FUNCTION_BLOCK FB_Roller_Door
VAR_INPUT
	// Inputs
    OpenBtn   : BOOL;
    CloseBtn  : BOOL;
    StopBtn   : BOOL;
    LS_Open   : BOOL;
    LS_Close  : BOOL;
END_VAR
VAR_OUTPUT
	// Outputs
    Motor_Up   : BOOL;
    Motor_Down : BOOL;
	Motor_Up_Reached:BOOL;
	Motor_Down_Reached:BOOL;
END_VAR
VAR
	// Internal states (latch)
    Opening : BOOL := FALSE;
    Closing : BOOL := FALSE;
END_VAR

// OPEN command
IF OpenBtn AND NOT LS_Open THEN
    Opening := TRUE;
    Closing := FALSE;
END_IF;
  
// CLOSE command
IF CloseBtn AND NOT LS_Close THEN
    Closing := TRUE;
    Opening := FALSE;
END_IF;
  
// STOP command
IF StopBtn THEN
    Opening := FALSE;
    Closing := FALSE;
END_IF;
  
// Limit conditions (auto stop)
IF LS_Open THEN
    Opening := FALSE;
END_IF;
 
IF LS_Close THEN
    Closing := FALSE;
END_IF;

// --- Outputs ---
Motor_Up := Opening AND NOT LS_Open;
Motor_Down := Closing AND NOT LS_Close;


Motor_Up_Reached := LS_Open;
Motor_Down_Reached := LS_Close;

END_FUNCTION_BLOCK

(* stored: Version 1.1.0.1, ProductVersion 3.1.4024.16
   POU FB_Roller_Door: Id {0eef03d8-0a87-4bfe-9819-8fb6545b98c6}, SpecialFunc None *)
